// TIA Portal V19 export
DATA_BLOCK "A0302_Bordatrice_RegolazioneFormato"   // DB74
// stored: InstanceOfName A0302_Bordatrice_RegolazioneFormato_FB, InstanceOfType FB
"A0302_Bordatrice_RegolazioneFormato_FB"
   // VAR_INPUT
   //    AreaInterface : "AreaInterface";
   //    ZSI : "udt_ZoneSafetyInterface";
   //    DSI_Formato : "udt_DeviceSafetyInterface";
   //    DSI_Cassetta : "udt_DeviceSafetyInterface";
   //    Cin : Struct
   //       LineSetup_Exe : Bool;
   //       OB30_High : Bool;
   //       Infeed_ON : Bool;
   //    END_STRUCT;
   //    DataIn : Struct
   //       PB_Passaggio01_Combo : "Ax_PB";
   //       PB_Passaggio02_Combo : "Ax_PB";
   //       PB_Passaggio03_Combo : "Ax_PB";
   //       PB_Passaggio04_Combo : "Ax_PB";
   //    END_STRUCT;
   // END_VAR
   // VAR_OUTPUT
   //    MachineInterface { ExternalAccessible := 'False'; ExternalVisible := 'False'; ExternalWritable := 'False'} : "MachineInterface";
   //    Cout : Struct
   //       OB30_High_Req : Bool;
   //       Infeed_ReqON : Bool;
   //       CtrlSafe_AX_M : Bool;
   //       SetUp_Bordatrice_Done : Array[1..9] of Bool;
   //    END_STRUCT;
   // END_VAR
   // VAR_IN_OUT
   //    Par_Machne : Struct
   //       Nervatura_Pos_Riposo : Real;
   //       Passaggio01_MaxDisallineamentoAXs : Real;
   //       Passaggio02_MaxDisallineamentoAXs : Real;
   //       Passaggio03_MaxDisallineamentoAXs : Real;
   //       Passaggio04_MaxDisallineamentoAXs : Real;
   //       AxD_AutoSpeed : Real;
   //    END_STRUCT;
   //    Par_Enc : Array[1..9] of "PosFbk_RTN";
   //    Par_D : Array[1..1] of "Positioning_DOL_Machine_Par";
   //    Par_M : Array[2..9] of "Positioning_MOL_Machine_Par";
   //    Pers_D : Array[1..1] of "Positioning_DOL_Machine_Pers_Data";
   //    Pers_M : Array[2..9] of "Positioning_MOL_Machine_Pers_Data";
   // END_VAR
   // VAR
   //    i : Int;
   //    Init_Done : Bool;
   //    HMI : Struct
   //       Passaggio01_Combo_TargetPos : Real;
   //       Passaggio02_Combo_TargetPos : Real;
   //       Passaggio03_Combo_TargetPos : Real;
   //       Passaggio04_Combo_TargetPos : Real;
   //    END_STRUCT;
   //    Warning : Struct
   //       Ax_D { S7_SetPoint := 'True'} : Array[1..1] of "Positioning_DOL_Machine_Wng";
   //       Ax_M : Array[1..9] of "Positioning_MOL_Machine_Wng";
   //       Passaggio01_MaxDisallineamentoAXs { S7_SetPoint := 'True'} : Bool;
   //       Passaggio02_MaxDisallineamentoAXs { S7_SetPoint := 'True'} : Bool;
   //       Passaggio03_MaxDisallineamentoAXs { S7_SetPoint := 'True'} : Bool;
   //       Passaggio04_MaxDisallineamentoAXs { S7_SetPoint := 'True'} : Bool;
   //    END_STRUCT;
   //    Alarm : Struct
   //       Enc : Array[1..9] of "PosFbk_Encoder_Alr";
   //       Ax_D { S7_SetPoint := 'True'} : Array[1..1] of "Positioning_DOL_Machine_Alr";
   //       Ax_M { S7_SetPoint := 'True'} : Array[1..9] of "Positioning_MOL_Machine_Alr";
   //    END_STRUCT;
   //    Sts : Struct
   //       UpdateSel : Int;
   //       Passaggio01 : Struct
   //          DeltaPos_OP_MOT : LReal;
   //          AxOP_Pause_Minus : Bool;
   //          AxOP_Pause_Plus : Bool;
   //          AxMOT_Pause_Minus : Bool;
   //          AxMOT_Pause_Plus : Bool;
   //       END_STRUCT;
   //       Passaggio02 : Struct
   //          DeltaPos_OP_MOT : LReal;
   //          AxOP_Pause_Minus : Bool;
   //          AxOP_Pause_Plus : Bool;
   //          AxMOT_Pause_Minus : Bool;
   //          AxMOT_Pause_Plus : Bool;
   //       END_STRUCT;
   //       Passaggio03 : Struct
   //          DeltaPos_OP_MOT : LReal;
   //          AxOP_Pause_Minus : Bool;
   //          AxOP_Pause_Plus : Bool;
   //          AxMOT_Pause_Minus : Bool;
   //          AxMOT_Pause_Plus : Bool;
   //       END_STRUCT;
   //       Passaggio04 : Struct
   //          DeltaPos_OP_MOT : LReal;
   //          AxOP_Pause_Minus : Bool;
   //          AxOP_Pause_Plus : Bool;
   //          AxMOT_Pause_Minus : Bool;
   //          AxMOT_Pause_Plus : Bool;
   //       END_STRUCT;
   //       TargetPos : Array[1..9] of Real;
   //    END_STRUCT;
   //    Ctrl : Struct
   //       OB30_High_Req : Bool;
   //       Passaggio01_Combo_MAN : Struct
   //          Minus : Bool;
   //          Plus : Bool;
   //          MoveToPos : Bool;
   //       END_STRUCT;
   //       Passaggio02_Combo_MAN : Struct
   //          Minus : Bool;
   //          Plus : Bool;
   //          MoveToPos : Bool;
   //       END_STRUCT;
   //       Passaggio03_Combo_MAN : Struct
   //          Minus : Bool;
   //          Plus : Bool;
   //          MoveToPos : Bool;
   //       END_STRUCT;
   //       Passaggio04_Combo_MAN : Struct
   //          Minus : Bool;
   //          Plus : Bool;
   //          MoveToPos : Bool;
   //       END_STRUCT;
   //    END_STRUCT;
   //    EncITF : Array[1..9] of "PosFbk_ITF";
   //    TOF_OB30_High { S7_SetPoint := 'True'} : TOF_TIME;
   //    Enc { S7_SetPoint := 'True'} : Array[1..9] of "PosFbk_SickAFM60";
   //    AX_D { S7_SetPoint := 'True'} : Array[1..1] of "Positioning_DOL_Machine_FB";
   //    AX_M { S7_SetPoint := 'True'} : Array[2..9] of "Positioning_MOL_Machine_FB";
   //    AUX : Struct
   //       PB_Passaggio01_Combo : Struct
   //          Minus : Bool;
   //          Plus : Bool;
   //          MoveToPos : Bool;
   //       END_STRUCT;
   //       PB_Passaggio02_Combo : Struct
   //          Minus : Bool;
   //          Plus : Bool;
   //          MoveToPos : Bool;
   //       END_STRUCT;
   //       PB_Passaggio03_Combo : Struct
   //          Minus : Bool;
   //          Plus : Bool;
   //          MoveToPos : Bool;
   //       END_STRUCT;
   //       PB_Passaggio04_Combo : Struct
   //          Minus : Bool;
   //          Plus : Bool;
   //          MoveToPos : Bool;
   //       END_STRUCT;
   //    END_STRUCT;
   // END_VAR
BEGIN
END_DATA_BLOCK
